FUNCTION_BLOCK earth_fault_1_3 (* Composite Function Block Type *)
  (* Standard: 61499-2 *)
  (* Version 0.0, 3/23/2016, gulzha, nxtControl GmbH, template *)
  PACKAGE Main;
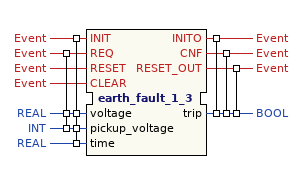
  EVENT_INPUT
    INIT WITH pickup_voltage, voltage, time; (* Initialization Request *)
    REQ WITH pickup_voltage, voltage; (* Normal Execution Request *)
    RESET;
    CLEAR;
  END_EVENT
  EVENT_OUTPUT
    INITO WITH trip; (* Initialization Confirm *)
    CNF WITH trip; (* Execution Confirmation *)
    RESET_OUT WITH trip;
  END_EVENT
  VAR_INPUT
    voltage : REAL;
    pickup_voltage : INT;
    time : REAL;
  END_VAR
  VAR_OUTPUT
    trip : BOOL;
  END_VAR
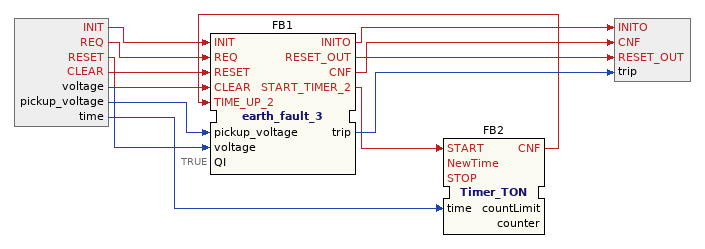
  FBS
    FB2 : Timer_TON;
    FB1 : earth_fault_3(QI := TRUE);
  END_FBS
  EVENT_CONNECTIONS
    INIT TO FB1.INIT;
    FB1.INITO TO INITO;
    REQ TO FB1.REQ;
    RESET TO FB1.RESET;
    FB1.RESET_OUT TO RESET_OUT;
    CLEAR TO FB1.CLEAR;
    FB1.CNF TO CNF;
    FB1.START_TIMER_2 TO FB2.START;
    FB2.CNF TO FB1.TIME_UP_2;
  END_CONNECTIONS
  DATA_CONNECTIONS
    pickup_voltage TO FB1.pickup_voltage;
    voltage TO FB1.voltage;
    FB1.trip TO trip;
    time TO FB2.time;
  END_CONNECTIONS
END_FUNCTION_BLOCK
